TYPE ST_MC_CMD :
STRUCT
	
bExe				: BOOL;
lrVelocity			: LREAL;
lrAcceleration		: LREAL;
lrDeceleration		: LREAL;
lrJerk				: LREAL;
lrDistance			: LREAL;
lrPosition			: LREAL;
EnuDirection		: MC_Direction;
EnuBufferMode		: MC_BufferMode;
EnuOptions			: ST_MoveOptions;

END_STRUCT
END_TYPE

(* stored: Version 1.1.0.1, ProductVersion 3.1.4024.12
   DUT ST_MC_CMD: Id {0847010a-9453-4a23-863f-4245417294d3} *)
